(* IEC 61131-3 sources: IRIS-Project/LASAL CONTROL SOFTWARE/LasalProject_2025_09_12/Class/Reset, 1 file *)

(* ---- Reset.st ---- *)
(*!
<Class
	Name               = "Reset"
	Revision           = "0.0"
	RealtimeTask       = "false"
	CyclicTask         = "true"
	DefCyclictime      = "100 ms"
	BackgroundTask     = "false"
	Sigmatek           = "false"
	OSInterface        = "false"
	HighPriority       = "false"
	Automatic          = "false"
	UpdateMode         = "Prescan"
	SharedCommandTable = "true"
	Objectsize         = "(550,120)">
	<Channels>
		<Server Name="ClassSvr" Visualized="false" Initialize="false" WriteProtected="true" Retentive="false"/>
		<Server Name="s_ResetT" Visualized="false" Initialize="false" WriteProtected="false" Retentive="false"/>
		<Client Name="c_ResetTimerDis" Required="true" Internal="false"/>
		<Client Name="c_ResetTimerIrr" Required="true" Internal="false"/>
		<Client Name="c_ResetTimerMov" Required="true" Internal="false"/>
	</Channels>
</Class>
*)
Reset : CLASS
  //Servers:
	ClassSvr 	: SvrChCmd_DINT;
	s_ResetT 	: SvrCh_DINT;
  //Clients:
	c_ResetTimerIrr 	: CltCh_DINT;
	c_ResetTimerMov 	: CltCh_DINT;
	c_ResetTimerDis 	: CltCh_DINT;
  //Variables:
  //Functions:

	FUNCTION VIRTUAL GLOBAL CyWork
		VAR_INPUT
			EAX 	: UDINT;
		END_VAR
		VAR_OUTPUT
			state (EAX) 	: UDINT;
		END_VAR;
  //Tables:
	FUNCTION @STD
		VAR_OUTPUT
			ret_code	: CONFSTATES;
		END_VAR;
	FUNCTION GLOBAL TAB @CT_;
END_CLASS;

FUNCTION VIRTUAL GLOBAL Reset::CyWork
	VAR_INPUT
		EAX 	: UDINT;
	END_VAR
	VAR_OUTPUT
		state (EAX) 	: UDINT;
	END_VAR

  if s_ResetT.Read() then
    c_ResetTimerDis.Write(input:=1);
    c_ResetTimerMov.Write(input:=1);
    c_ResetTimerIrr.Write(input:=1);
  else
    c_ResetTimerDis.Write(input:=0);
    c_ResetTimerMov.Write(input:=0);
    c_ResetTimerIrr.Write(input:=0);
  end_if;

	state := READY;

END_FUNCTION
